// Mitsubishi GX Works2 project: 계산기   PLC: Q02/Q02H

PROGRAM MAIN
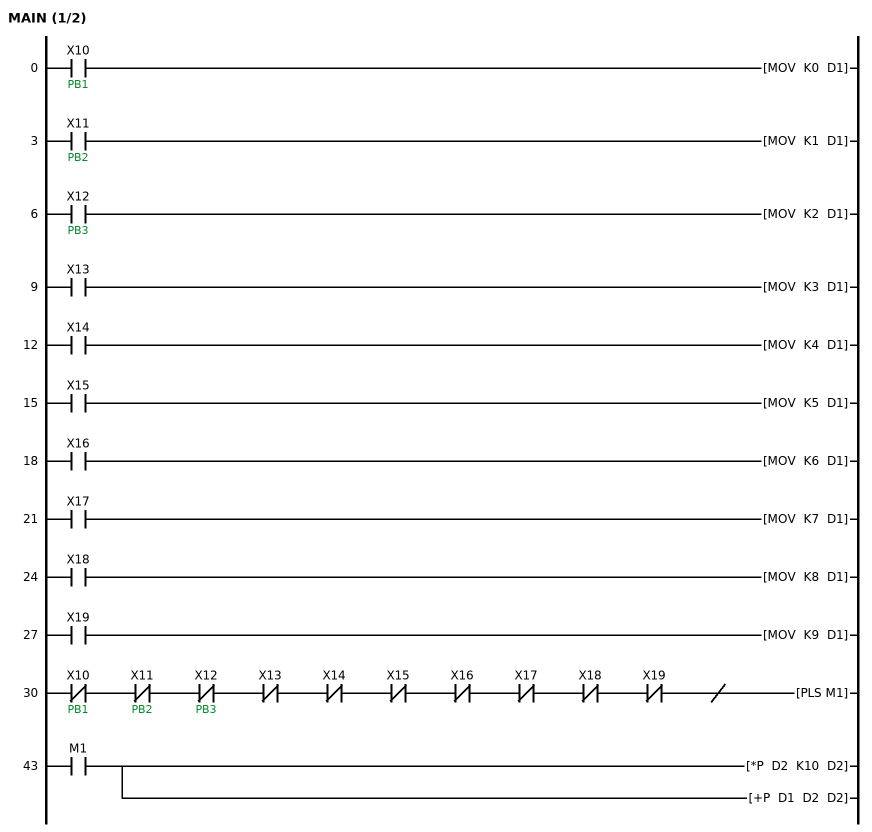
0     LD      X10  ; PB1
      MOV     K0 D1
3     LD      X11  ; PB2
      MOV     K1 D1
6     LD      X12  ; PB3
      MOV     K2 D1
9     LD      X13
      MOV     K3 D1
12    LD      X14
      MOV     K4 D1
15    LD      X15
      MOV     K5 D1
18    LD      X16
      MOV     K6 D1
21    LD      X17
      MOV     K7 D1
24    LD      X18
      MOV     K8 D1
27    LD      X19
      MOV     K9 D1
30    LDI     X10  ; PB1
      ANI     X11  ; PB2
      ANI     X12  ; PB3
      ANI     X13
      ANI     X14
      ANI     X15
      ANI     X16
      ANI     X17
      ANI     X18
      ANI     X19
      INV
      PLS     M1
43    LD      M1
      *P      D2 K10 D2
      +P      D1 D2 D2
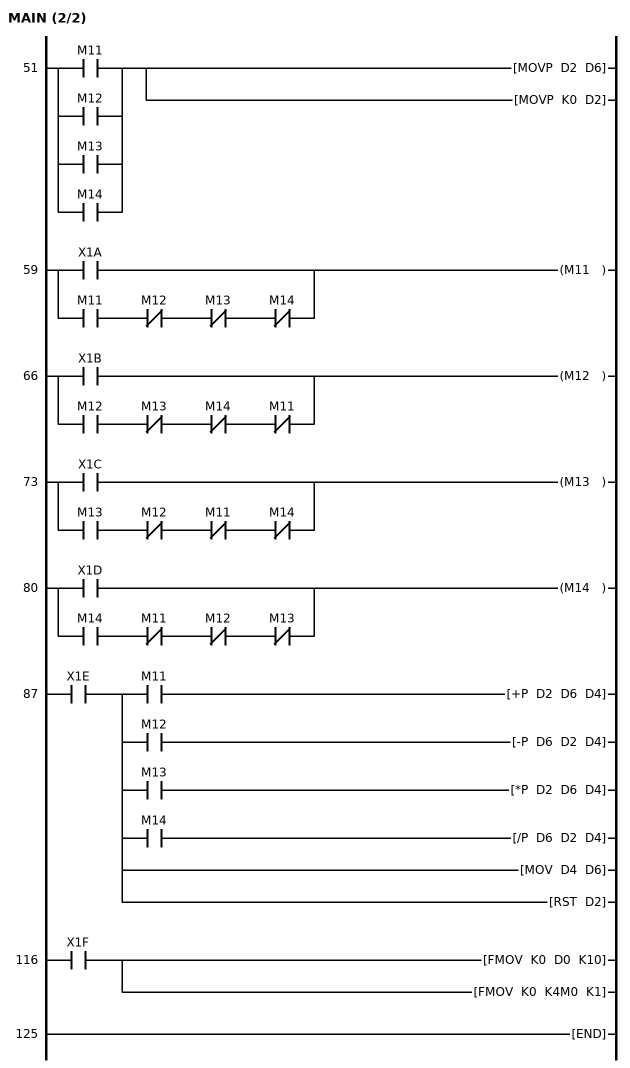
51    LD      M11
      OR      M12
      OR      M13
      OR      M14
      MOVP    D2 D6
      MOVP    K0 D2
59    LD      X1A
      LD      M11
      ANI     M12
      ANI     M13
      ANI     M14
      ORB
      OUT     M11
66    LD      X1B
      LD      M12
      ANI     M13
      ANI     M14
      ANI     M11
      ORB
      OUT     M12
73    LD      X1C
      LD      M13
      ANI     M12
      ANI     M11
      ANI     M14
      ORB
      OUT     M13
80    LD      X1D
      LD      M14
      ANI     M11
      ANI     M12
      ANI     M13
      ORB
      OUT     M14
87    LD      X1E
      MPS
      AND     M11
      +P      D2 D6 D4
      MRD
      AND     M12
      -P      D6 D2 D4
      MRD
      AND     M13
      *P      D2 D6 D4
      MRD
      AND     M14
      /P      D6 D2 D4
      MPP
      MOV     D4 D6
      RST     D2
116   LD      X1F
      FMOV    K0 D0 K10
      FMOV    K0 K4M0 K1
125   END
END_PROGRAM

// device comments not shown above
X0  ; 공급_후
X1  ; 공급_전
X2  ; 드릴_상
X3  ; 드릴_하
X4  ; 송출_후
X5  ; 송출_전
X6  ; 배출_후
X7  ; 배출_전
X8  ; 매거진
X9  ; 비금속
X0A  ; 금속
Y20  ; 공급_전
Y21  ; 공급_후
Y22  ; 드릴_하강
Y23  ; 송출_전
Y24  ; 송출_후
Y25  ; 배출_전
Y26  ; 배출_후
Y27  ; 컨베어
Y28  ; 가공드
Y29  ; 적색
Y2A  ; 황색
Y2B  ; 녹색
